FUNCTION_BLOCK FB_Alarm EXTENDS FB_TcAlarm
VAR_INPUT
	evtEntry		: TcEventEntry;
	bEvt			: BOOL;
	bClear			: BOOL;
END_VAR
VAR_OUTPUT
END_VAR
VAR
	r_TrigEvt		: r_Trig;
	r_TrigClr		: r_Trig;
	b_Init			: BOOL := TRUE;
	b_mem			: BOOL;
END_VAR

IF b_Init THEN
	SUPER^.CreateEx(evtEntry, TRUE, 0);
END_IF

r_TrigEvt(CLK:=bEvt);
r_TrigClr(CLK:=bClear);

IF bEvt THEN
	SUPER^.Raise(0);
END_IF

//IF r_TrigClr.Q THEN
//	SUPER^.Clear(0, FALSE);
//END_IF

END_FUNCTION_BLOCK

(* stored: Version 1.1.0.1, ProductVersion 3.1.4024.12
   POU FB_Alarm: Id {e29bb0e6-c248-48d4-ac6b-27b396e84f7c}, SpecialFunc None *)
